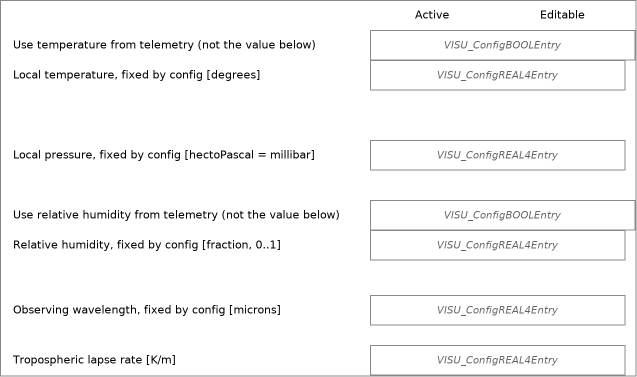
VISUALIZATION VISU_AxesConfig_LocalConditions  // 637x377
VAR_IN_OUT
    active : AxesLocalConditionsConfig;
    editable : AxesLocalConditionsConfig;
END_VAR
    Label (370,5 125x20), "Active"
    Label (500,5 125x20), "Editable"
    Label (10,30 360x30), "Use temperature from telemetry (not the value below)"
    Frame (370,30 265x30)
        shows VISU_ConfigBOOLEntry(active := active.useTemperatureFromSensors, editable := editable.useTemperatureFromSensors)
    Label (10,60 360x30), "Local temperature, fixed by config [degrees]"
    Frame (370,60 255x30)
        shows VISU_ConfigREAL4Entry(active := active.configuredTemperature, editable := editable.configuredTemperature)
    Label (10,140 360x30), "Local pressure, fixed by config [hectoPascal = millibar]"
    Frame (370,140 255x30)
        shows VISU_ConfigREAL4Entry(active := active.configuredPressure, editable := editable.configuredPressure)
    Label (10,230 360x30), "Relative humidity, fixed by config [fraction, 0..1]"
    Label (10,200 360x30), "Use relative humidity from telemetry (not the value below)"
    Frame (370,200 265x30)
        shows VISU_ConfigBOOLEntry(active := active.useRelativeHumidityFromSensors, editable := editable.useRelativeHumidityFromSensors)
    Frame (370,230 255x30)
        shows VISU_ConfigREAL4Entry(active := active.configuredRelativeHumidity, editable := editable.configuredRelativeHumidity)
    Label (10,295 360x30), "Observing wavelength, fixed by config [microns]"
    Frame (370,295 255x30)
        shows VISU_ConfigREAL4Entry(active := active.configuredObservingWavelength, editable := editable.configuredObservingWavelength)
    Label (10,345 360x30), "Tropospheric lapse rate [K/m]"
    Frame (370,345 255x30)
        shows VISU_ConfigREAL4Entry(active := active.troposphericLapseRate, editable := editable.troposphericLapseRate)
END_VISUALIZATION

(* stored: Version 1.1.0.1, ProductVersion 3.1.4019.2
   Visu VISU_AxesConfig_LocalConditions: Id {6bf78346-d66a-4c11-a5a0-6645228648b7} *)
